IF i > len_active_pumps  THEN
	i := len_active_pumps;
ELSIF i < 1 THEN
	i := 1;
END_IF;
END_ACTION
ACTION check_active_pumps:
pumps[1] := get_active(info_invertor_drive1);
pumps[2] := get_active(info_invertor_drive2);
pumps[3] := get_active(info_invertor_drive3);
pumps[4] := get_active(info_invertor_drive4);
pumps[5] := get_active(info_invertor_drive5);
pumps[6] := get_active(info_invertor_drive6);
pumps[7] := get_active(info_invertor_drive7);
pumps[8] := get_active(info_invertor_drive8);

len_pumps := len_bool_array(pumps);  (* get en input pumps array. *)
index_active_pumps := index_bool_array(pumps);  (* get indexes active pumps. *)
len_active_pumps := len_int_array(index_active_pumps);  (* get len active pumps. *)

index_pivot := index_element_in_int_array(pivot, index_active_pumps); (* get index pivot.*)
END_ACTION
ACTION check_pivot:
error_code := 3;
error_message := 'pivot pump not excpect int more 0.';
END_ACTION
ACTION get_info_message:
IF enable AND error_message = 'GOOD' THEN
	info_cascade.pivot := pivot;
	info_cascade.error_message := error_message;
	info_cascade.cascade_pump1 := cascade_pumps[1];
	info_cascade.cascade_pump2 := cascade_pumps[2];
	info_cascade.cascade_pump3 := cascade_pumps[3];
	info_cascade.cascade_pump4 := cascade_pumps[4];
	info_cascade.cascade_pump5 := cascade_pumps[5];
	info_cascade.cascade_pump6 := cascade_pumps[6];
	info_cascade.cascade_pump7 := cascade_pumps[7];
	info_cascade.cascade_pump8 := cascade_pumps[8];
	info_cascade.error_code := error_code;
ELSE
	info_cascade.pivot := index_pivot;
	info_cascade.error_code := error_code;
	info_cascade.error_message := error_message;
	cascade_pumps[1].cascade_pump := FALSE;
	cascade_pumps[2].cascade_pump := FALSE;
	cascade_pumps[3].cascade_pump := FALSE;
	cascade_pumps[4].cascade_pump := FALSE;
	cascade_pumps[5].cascade_pump := FALSE;
	cascade_pumps[6].cascade_pump := FALSE;
	cascade_pumps[7].cascade_pump := FALSE;
	cascade_pumps[8].cascade_pump := FALSE;
	info_cascade.cascade_pump1 := cascade_pumps[1];
	info_cascade.cascade_pump2 := cascade_pumps[2];
	info_cascade.cascade_pump3 := cascade_pumps[3];
	info_cascade.cascade_pump4 := cascade_pumps[4];
	info_cascade.cascade_pump5 := cascade_pumps[5];
	info_cascade.cascade_pump6 := cascade_pumps[6];
	info_cascade.cascade_pump7 := cascade_pumps[7];
	info_cascade.cascade_pump8 := cascade_pumps[8];
END_IF;
END_ACTION

(* POU function/methods_8_array/len_bool_array, ST *)
FUNCTION len_bool_array : INT

VAR_INPUT
	list: ARRAY [1..8] OF BOOL;
END_VAR

VAR
	size: INT := 8;
	cnt:INT := 0;
	i: INT;
END_VAR
FOR i := 1 TO size DO
	IF list[i] THEN
		cnt := cnt + 1;
	END_IF;
END_FOR;

IF i > 8 THEN
	i := 1;
END_IF;

len_bool_array := cnt;
END_FUNCTION

(* POU function/methods_8_array/index_bool_array, ST *)
FUNCTION index_bool_array : ARRAY [1..8] OF INT

VAR_INPUT
	list:ARRAY [1..8] OF BOOL;
END_VAR

VAR
	size:INT := 8;
	i: INT;
	cnt:INT := 1;
	index:ARRAY [1..8] OF INT := 8(0);
END_VAR
FOR i:= 1 TO size DO
	IF list[i] THEN
		index[cnt] := i;
		cnt := cnt + 1;
	END_IF;
END_FOR;

index_bool_array := index;
END_FUNCTION

(* POU function/methods_8_array/len_int_array, ST *)
FUNCTION len_int_array : INT

VAR_INPUT
	list: ARRAY [1..8] OF INT;
END_VAR

VAR
	size: INT:=8;
	cnt:INT:=0;
	i: INT;
END_VAR
FOR i:=1 TO size DO
	IF INT_TO_BOOL(list[i]) THEN
		cnt:=cnt + 1;
	END_IF;
END_FOR;

IF i > 8 THEN
	i:=1;
END_IF;

len_int_array:=cnt;
END_FUNCTION

(* POU function/methods_8_array/index_element_in_int_array, ST *)
FUNCTION index_element_in_int_array : INT

VAR_INPUT
	element:INT;
	list:ARRAY [1..8] OF  INT;
END_VAR

VAR
	size: INT := 8;
	i: INT;
	index: INT := 1;
END_VAR
IF element_in_int_array(element, list) THEN
	FOR i := 1 TO size DO
		IF list[i]=element THEN
			index := i;
			i := 8;
		END_IF;
	END_FOR;
	index_element_in_int_array := index;
ELSE
	index_element_in_int_array := 0;
END_IF;
END_FUNCTION

(* POU function/methods_8_array/element_in_int_array, ST *)
FUNCTION element_in_int_array : BOOL

VAR_INPUT
	element:INT;
	list: ARRAY [1..8] OF INT;
END_VAR

VAR
	size: INT := 8;
	i: INT;
	is_true:BOOL := FALSE;
END_VAR
FOR i := 1 TO size DO
	IF list[i]=element THEN
		is_true := TRUE;
	END_IF;
END_FOR;

element_in_int_array := is_true;
END_FUNCTION

(* POU mode_selector/Cascade_Cycle_Selector, ST *)
FUNCTION_BLOCK Cascade_Cycle_Selector
(* Function block implementation working mode selector. *)

VAR_INPUT
    cascade: BOOL; (* enable/disable *)
    cycle: BOOL; (* enable/disable *)
    single: BOOL; (* enable/disable *)
    info_single: classInfoSingle;
    info_cycle: classInfoCycle;
    info_cascade: classInfoCascade;
END_VAR

VAR_OUTPUT
    mode_selector_error: WORD;
    start_pump1: BOOL := FALSE;
    start_pump2: BOOL := FALSE;
    start_pump3: BOOL := FALSE;
    start_pump4: BOOL := FALSE;
    start_pump5: BOOL := FALSE;
    start_pump6: BOOL := FALSE;
    start_pump7: BOOL := FALSE;
    start_pump8: BOOL := FALSE;
END_VAR

VAR
    message: STRING(79);
    flag_mode: INT;
	error_code: WORD;
END_VAR
IF cascade AND NOT cycle AND NOT single THEN
    flag_mode := 2;
    message := 'Cascade mode selected'; (* Выбран каскадный режим работы. *)
ELSIF cycle AND NOT cascade AND NOT single THEN
    flag_mode := 1;
    message := 'Cycle mode selected'; (* Выбран циклический режим работы *)
ELSIF single AND NOT cycle AND NOT cascade THEN
    flag_mode := 0;
    message := 'Single mode selected'; (* Выбран режим работы одного насоса *) 
ELSE
    flag_mode := -1;
    error_code := 7;
    message := 'Select any one working mode!'; (* Выберите один режим работы! *)
END_IF;

IF flag_mode = 0 THEN
    start_pump1 := get_pump_in_single(info_single, 1);
    start_pump2 := get_pump_in_single(info_single, 2);
    start_pump3 := get_pump_in_single(info_single, 3);
    start_pump4 := get_pump_in_single(info_single, 4);
    start_pump5 := get_pump_in_single(info_single, 5);
    start_pump6 := get_pump_in_single(info_single, 6);
    start_pump7 := get_pump_in_single(info_single, 7);
    start_pump8 := get_pump_in_single(info_single, 8);
    mode_selector_error := info_single.error_code;
ELSIF flag_mode = 1 THEN
    start_pump1 := get_pump_in_cycle(info_cycle, 1);
    start_pump2 := get_pump_in_cycle(info_cycle, 2);
    start_pump3 := get_pump_in_cycle(info_cycle, 3);
    start_pump4 := get_pump_in_cycle(info_cycle, 4);
    start_pump5 := get_pump_in_cycle(info_cycle, 5);
    start_pump6 := get_pump_in_cycle(info_cycle, 6);
    start_pump7 := get_pump_in_cycle(info_cycle, 7);
    start_pump8 := get_pump_in_cycle(info_cycle, 8);
    mode_selector_error := info_cycle.error_code;
ELSIF flag_mode = 2 THEN
    start_pump1 := get_pump_in_cascade(info_cascade, 1);
    start_pump2 := get_pump_in_cascade(info_cascade, 2);
    start_pump3 := get_pump_in_cascade(info_cascade, 3);
    start_pump4 := get_pump_in_cascade(info_cascade, 4);
    start_pump5 := get_pump_in_cascade(info_cascade, 5);
    start_pump6 := get_pump_in_cascade(info_cascade, 6);
    start_pump7 := get_pump_in_cascade(info_cascade, 7);
    start_pump8 := get_pump_in_cascade(info_cascade, 8);
    mode_selector_error := info_cascade.error_code;
ELSE
    start_pump1 := FALSE;
    start_pump2 := FALSE;
    start_pump3 := FALSE;
    start_pump4 := FALSE;
    start_pump5 := FALSE;
    start_pump6 := FALSE;
    start_pump7 := FALSE;
    start_pump8 := FALSE;
    mode_selector_error := error_code;
END_IF;
END_FUNCTION_BLOCK

(* POU single_mode/get_pump_in_single, ST *)
FUNCTION get_pump_in_single : BOOL
(* Function get status pump in information single mode *)

VAR_INPUT
    info_single: classInfoSingle;
    pump_number: INT;
END_VAR
IF pump_number = info_single.pivot_pump THEN
    get_pump_in_single := info_single.start_pump;
ELSE
    get_pump_in_single := FALSE;
END_IF;
END_FUNCTION

(* POU cycle_mode/get_pump_in_cycle, ST *)
FUNCTION get_pump_in_cycle : BOOL (*ï¿½ï¿½ï¿½ï¿½ï¿½ï¿½ï¿½ ï¿½ï¿½ï¿½ï¿½ï¿½ï¿½ï¿½ï¿½ï¿½ï¿½ï¿½ï¿½ ï¿½ï¿½ï¿½ï¿½ ï¿½ï¿½ï¿½ï¿½ï¿½ï¿½ ï¿½ï¿½ï¿½ï¿½ï¿½ï¿½ï¿½ï¿½ï¿½ï¿½ ï¿½ï¿½ï¿½ï¿½ï¿½ï¿½ *)

VAR_INPUT
	info_cycle:classInfoCycle;
	pump_number:SINT;
END_VAR
IF pump_number=info_cycle.pump_number THEN
	get_pump_in_cycle:=info_cycle.run_timer;
ELSE
	get_pump_in_cycle:=FALSE;
END_IF;
END_FUNCTION

(* POU cascade_mode/get_pump_in_cascade, ST *)
FUNCTION get_pump_in_cascade : BOOL

VAR_INPUT
	info:classInfoCascade;
	number_pump:INT;
END_VAR

VAR
	pumps:ARRAY[1..8] OF classInfoCascadePump;
END_VAR
IF info.pivot = number_pump THEN
	get_pump_in_cascade:=TRUE;
ELSE
	pumps[1]:=info.cascade_pump1;
	pumps[2]:=info.cascade_pump2;
	pumps[3]:=info.cascade_pump3;
	pumps[4]:=info.cascade_pump4;
	pumps[5]:=info.cascade_pump5;
	pumps[6]:=info.cascade_pump6;
	pumps[7]:=info.cascade_pump7;
	pumps[8]:=info.cascade_pump8;

	get_pump_in_cascade:=pumps[number_pump].cascade_pump;
END_IF;
END_FUNCTION

(* POU DanfossKPI/Kpi, ST *)
FUNCTION_BLOCK Kpi

VAR_INPUT
	input:BOOL;  (* ï¿½ï¿½ï¿½ï¿½ï¿½ï¿½ï¿½ï¿½ ï¿½ï¿½ ï¿½ï¿½ï¿½ï¿½ï¿½ *)
END_VAR

VAR_OUTPUT
	NC:BOOL; (* normal close �2 *)
	NO:BOOL; (* normal open �4 *)
END_VAR

VAR
END_VAR
NC:=NOT input;
NO:=input;
END_FUNCTION_BLOCK

(* POU Alarm_manager_error/ALARM_MANAGER, ST *)
FUNCTION_BLOCK ALARM_MANAGER
(* Function block handle alarm. *)

VAR_INPUT
    low_pressure_input: BOOL;
    high_pressure_out: BOOL;
    external_alarm_invertor_drive_code: WORD;
    input_pressure_error_code: WORD;
    out_pressure_error_code: WORD;
    mode_selector_error: WORD;
END_VAR

VAR_OUTPUT
    alarm_on: BOOL := TRUE;
    error_code_alarm: WORD;
    error_message: STRING(79);
END_VAR
IF low_pressure_input THEN
    error_code_alarm := 1;
ELSIF high_pressure_out THEN
    error_code_alarm := 2;
ELSIF external_alarm_invertor_drive_code > 0 THEN
    error_code_alarm := external_alarm_invertor_drive_code;
ELSIF input_pressure_error_code > 0 THEN
    error_code_alarm := input_pressure_error_code;
ELSIF out_pressure_error_code > 0 THEN
    error_code_alarm := input_pressure_error_code;
ELSIF mode_selector_error > 0 THEN
    error_code_alarm := mode_selector_error;
ELSE
    error_code_alarm := 0;
END_IF;

IF error_code_alarm <> 0 THEN
    alarm_on := TRUE;
    error_message := get_alarm_message(error_code_alarm);
ELSE
    alarm_on := FALSE;
END_IF;
END_FUNCTION_BLOCK

(* POU Alarm_manager_error/get_alarm_message, ST *)
FUNCTION get_alarm_message : STRING(79)
(* Function return message alarm of error_code *)

VAR_INPUT
    code_error: WORD;
END_VAR

VAR
    error_message: STRING(79);
END_VAR
IF code_error = 0
	THEN error_message := 'Аварий нет.'; (* Measure good *)
ELSIF code_error = 1
    THEN error_message := 'Низкое давление на входе! (защита по сухому ходу)'; (* low input pressure!*)
ELSIF code_error = 2 
    THEN error_message := 'Высокое давление на выходе! (защита по превышению давления)'; (* high output pressure! *)
ELSIF code_error = 3
    THEN error_message := 'В каскадном режиме должен быть выбран опорный насос.'; (* Pivot cascade pump not expected int more 0! *)
ELSIF code_error = 4
    THEN error_message := 'В каскадном режиме должно быть более одного активного насоса.'; (* Cascade mode excpected more one active pumps, but got less! *)
ELSIF code_error = 5
    THEN error_message := 'В каскадном режиме выбранный опорный насос не активен.'; (* Cascade pivot pump not active! *)
ELSIF code_error = 6
    THEN error_message := 'В одиночном режиме выбранный насос не активени.'; (* Single mode select pump is not active! *)
ELSIF code_error = 7
    THEN error_message := 'Выберите только один режим работы станции.'; (* Select any one working mode! *)
ELSIF code_error = 8
    THEN error_message := 'Внешняя авария частотного преобразователя №1'; (* External alarm invertor drive 1 *)
ELSIF code_error = 9
    THEN error_message := 'Внешняя авария частотного преобразователя №2'; (* External alarm invertor drive 2. *)
ELSIF code_error = 10
    THEN error_message := 'Внешняя авария частотного преобразователя №3'; (* External alarm invertor drive 3. *)
ELSIF code_error = 11
    THEN error_message := 'Внешняя авария частотного преобразователя №4'; (* External alarm invertor drive 4. *)
ELSIF code_error = 12
    THEN error_message := 'Внешняя авария частотного преобразователя №5'; (* External alarm invertor drive 5. *)
ELSIF code_error = 13
    THEN error_message := 'Внешняя авария частотного преобразователя №6'; (* External alarm invertor drive 6. *)
ELSIF code_error = 14
    THEN error_message := 'Внешняя авария частотного преобразователя №7'; (* External alarm invertor drive 7. *)
ELSIF code_error = 15
    THEN error_message := 'Внешняя авария частотного преобразователя №8'; (* External alarm invertor drive 8. *)
ELSIF code_error = 61440
	THEN error_message := 'Ошибка  AQ. Значение заведомо неверно.'; (* Value bad! *)
ELSIF code_error = 61446
	THEN error_message := 'Ошибка AQ.  Данные не готовы. Ждите результатов первого измеорения. '; (* Data info not complete! Wait first measuring. *)
ELSIF code_error = 61447
	THEN error_message := 'Ошибка AQ. Датчик отключен.'; (* Sensor off. *)
ELSIF code_error = 61448
	THEN error_message := 'Ошибка AQ. Велика температура свободных концов ТП.'; (* Temperature free ends of termosensor high. *)
ELSIF code_error = 61449
	THEN error_message := 'Ошибка AQ. Мала температура свободных концов ТП.'; (* Temperature free ends of termosensor low. *)
ELSIF code_error = 61450
	THEN error_message := 'Ошибка AQ. Измеренное значение слишком велико!'; (* Measured value too more. *)
ELSIF code_error = 61451
	THEN error_message := 'Ошибка AQ. Измеренное значение слишком мало!'; (* Measured value too less. *)
ELSIF code_error = 61452
	THEN error_message := 'Ошибка AQ.  Короткое замыкание датчика.'; (* Short circuit of sensor. *)
ELSIF code_error = 61453
	THEN error_message := 'Ошибка AQ. Обрыв датчика.'; (* Sensor breaking. *)
ELSIF code_error = 61454
	THEN error_message := 'Ошибка AQ. Отсутствие связи с АЦП.'; (* Failure connection with DAC. *)
ELSIF code_error = 61455
	THEN error_message := 'Ошибка AQ. Некорректный калибровочный коэффициент.'; (* Uncorrect calibrate rate. *)
ELSE
	error_message := 'Error not Found';
END_IF

get_alarm_message := error_message;
    
END_FUNCTION

(* POU Alarm_manager_error/external_alarm_invertor_drive, ST *)
FUNCTION_BLOCK external_alarm_invertor_drive
(* Function block return code error external alarm of invertor drives in PLC110-32m2 *)

VAR_INPUT
    status_inputs: classPLC32m2StatusInputs;
    number_di_alarm_id1: INT := 0;
    number_di_alarm_id2: INT := 0;
    number_di_alarm_id3: INT := 0;
    number_di_alarm_id4: INT := 0;
    number_di_alarm_id5: INT := 0;
    number_di_alarm_id6: INT := 0;
    number_di_alarm_id7: INT := 0;
    number_di_alarm_id8: INT := 0;
END_VAR

VAR_OUTPUT
    error_code_alarm: WORD;
END_VAR

VAR
    check_alarm: INT;
    error_code: WORD;
    i: INT;
    number_di_alarm: ARRAY [1..8] OF INT;
    pump_alarm: ARRAY [1..8] OF BOOL;
    index_alarm: ARRAY [1..8] OF INT;
END_VAR
number_di_alarm[1] := number_di_alarm_id1;
number_di_alarm[2] := number_di_alarm_id2;
number_di_alarm[3] := number_di_alarm_id3;
number_di_alarm[4] := number_di_alarm_id4;
number_di_alarm[5] := number_di_alarm_id5;
number_di_alarm[6] := number_di_alarm_id6;
number_di_alarm[7] := number_di_alarm_id7;
number_di_alarm[8] := number_di_alarm_id8;

FOR i := 1 TO 8 DO
    IF number_di_alarm[i] > 0 THEN
        pump_alarm[i] := get_di(number_di_alarm[i], status_inputs);
    ELSE
        pump_alarm[i] := FALSE;
    END_IF;
END_FOR;

check_alarm := len_bool_array(pump_alarm);
IF check_alarm > 0  THEN
    index_alarm := index_bool_array(pump_alarm);
    error_code := 7 + index_alarm[1];
ELSE
    error_code := check_alarm;
END_IF;

error_code_alarm := error_code;
END_FUNCTION_BLOCK

(* POU PLC110_32/get_di, ST *)
FUNCTION get_di : BOOL

VAR_INPUT
	input_number:INT;
	status_inputs:classPLC32m2StatusInputs;
END_VAR

VAR
	in_f:classDiscreteInputByte;
	in_s:classDiscreteInputByte;
	di_list:ARRAY[1..17] OF BOOL;
END_VAR
in_f:=status_inputs.discrete_inputs.first_byte;
in_s:=status_inputs.discrete_inputs.second_byte;

di_list[1]:=in_f.Bit1;
di_list[2]:=in_f.Bit2;
di_list[3]:=in_f.Bit3;
di_list[4]:=in_f.Bit4;
di_list[5]:=in_f.Bit5;
di_list[6]:=in_f.Bit6;
di_list[7]:=in_f.Bit7;
di_list[8]:=in_f.Bit8;

di_list[9]:=in_s.Bit1;
di_list[10]:=in_s.Bit2;
di_list[11]:=in_s.Bit3;
di_list[12]:=in_s.Bit4;
di_list[13]:=in_s.Bit5;
di_list[14]:=in_s.Bit6;
di_list[15]:=in_s.Bit7;
di_list[16]:=in_s.Bit8;

get_di:=di_list[input_number];
END_FUNCTION

(* POU PressureSensor_4_20ma/SetCurrentSensorPressure_4_20, ST *)
FUNCTION_BLOCK SetCurrentSensorPressure_4_20

VAR_INPUT
	min_measure_range:REAL:=0;
	max_measure_range:REAL:=16;
	min_current_range:REAL:=4;
	max_current_range:REAL:=20;
END_VAR

VAR_OUTPUT
	sensor_params:classSetPressureSensor4_20;
END_VAR
sensor_params.min_measure_range := min_measure_range;
sensor_params.max_measure_range := max_measure_range;
sensor_params.min_current_range := min_current_range;
sensor_params.max_current_range := max_current_range;
END_FUNCTION_BLOCK

(* POU Invertor_Drive/get_aout_current_in_info, ST *)
FUNCTION get_aout_current_in_info : REAL

VAR_INPUT
	info_invertor_drive:classInfoInvertorDrive;
END_VAR
get_aout_current_in_info:=info_invertor_drive.aout_frequency;
END_FUNCTION

(* POU Invertor_Drive/get_run_in_info, ST *)
FUNCTION get_run_in_info : BOOL

VAR_INPUT
	info_invertor_drive:classInfoInvertorDrive;
END_VAR
get_run_in_info:=info_invertor_drive.run ;
END_FUNCTION

(* POU Invertor_Drive/get_reset_faults, ST *)
FUNCTION get_reset_faults : BOOL

VAR_INPUT
    info: classInfoInvertorDrive; (* Comment *)
END_VAR
get_reset_faults := info.reset_fault;
END_FUNCTION

(* POU MB110_8.A/get_channel_current_value, ST *)
FUNCTION get_channel_current_value : REAL
(* ï¿½ï¿½ï¿½ï¿½ï¿½ï¿½ï¿½ ï¿½ï¿½ï¿½ï¿½ï¿½ï¿½ï¿½ï¿½ï¿½ï¿½ï¿½ï¿½ï¿½ InfoMessage ï¿½ï¿½ AnalogInputsModule  ï¿½ ï¿½ï¿½ï¿½ï¿½ï¿½ï¿½ï¿½ ï¿½ï¿½ ï¿½ï¿½ï¿½ï¿½ï¿½ï¿½ï¿½ ï¿½ï¿½ï¿½ï¿½ï¿½ï¿½ ï¿½ï¿½ï¿½ï¿½ï¿½ï¿½ï¿½ï¿½ ï¿½ï¿½ï¿½ï¿½ *)

VAR_INPUT
	ch_number:INT;
	Ain_info:classInfoAnalogInputModule;
END_VAR

VAR
	list_value : ARRAY [1..8] OF REAL;
END_VAR
list_value[1] := Ain_info.channel1.current_value;
list_value[2] := Ain_info.channel2.current_value;
list_value[3] := Ain_info.channel3.current_value;
list_value[4] := Ain_info.channel4.current_value;
list_value[5] := Ain_info.channel5.current_value;
list_value[6] := Ain_info.channel6.current_value;
list_value[7] := Ain_info.channel7.current_value;
list_value[8] := Ain_info.channel8.current_value;

get_channel_current_value := list_value[ch_number];
END_FUNCTION

(* POU function/hms_to_time, ST *)
FUNCTION hms_to_time : TIME
VAR_INPUT
	hours: WORD;
	minutes: WORD;
	seconds: WORD;
END_VAR
VAR
	MILLISECONDS_IN_HOUR: DWORD := 3600000;
	MILLISECONDS_IN_MINUTE: DWORD := 60000;
	MILLISECONDS_IN_SECOND: DWORD := 1000;
END_VAR
hms_to_time := DWORD_TO_TIME(
    (WORD_TO_DWORD(hours) * MILLISECONDS_IN_HOUR)
    + (WORD_TO_DWORD(minutes) * MILLISECONDS_IN_MINUTE)
    + (WORD_TO_DWORD(seconds) * MILLISECONDS_IN_SECOND)
);
END_FUNCTION

(* POU cascade_mode/get_auto_in_cascade, ST *)
FUNCTION get_auto_in_cascade : BOOL

VAR_INPUT
	info:classInfoCascade;
	number_pump:INT;
END_VAR
IF info.pivot=number_pump THEN
	get_auto_in_cascade:=TRUE;
ELSE
	get_auto_in_cascade:=FALSE;
END_IF;
END_FUNCTION

(* POU PLC110_32/get_fdi, ST *)
FUNCTION get_fdi : BOOL
(* ï¿½ï¿½ï¿½ï¿½ï¿½ï¿½ï¿½ï¿½ï¿½ï¿½ï¿½ï¿½ï¿½ ï¿½ï¿½ ï¿½ï¿½ï¿½ï¿½ï¿½ï¿½ï¿½ ï¿½ï¿½ï¿½ï¿½ï¿½ï¿½ ï¿½ï¿½ï¿½ï¿½ï¿½ï¿½ ï¿½ï¿½ï¿½ï¿½ï¿½ï¿½ï¿½ï¿½ï¿½ FDI *)
VAR_INPUT
	num:INT;
	status_inputs:classPLC32m2StatusInputs;
END_VAR

VAR
	fdi_list:ARRAY [1..2] OF BOOL;
END_VAR
fdi_list[1]:=status_inputs.fast_inputs.Bit1;
fdi_list[2]:=status_inputs.fast_inputs.Bit2;

get_fdi:=fdi_list[num];
END_FUNCTION

(* POU Invertor_Drive/get_frequency_in_info, ST *)
FUNCTION get_frequency_in_info : REAL
VAR_INPUT
	info_invertor_drive:classInfoInvertorDrive;
END_VAR
VAR
END_VAR
get_frequency_in_info:=info_invertor_drive.frequency;
END_FUNCTION
